   ELSE
       // ruch czarnych
       // 
       //ruch po skosie 
       #wykonuj_petle := TRUE;
       #poz_temp := #hetman.pozycja;
       WHILE #wykonuj_petle DO
           #poz_temp.x += 1;
           #poz_temp.y += 1;
           IF "sprawdz_czy_na_szachownicy"(#poz_temp) = true THEN
               IF "sprawdz_czy_wolne"(pozycja := #poz_temp, szachownica := #szachownica) = true THEN
                   IF "sprawdz_czy_ruch_możliwy"(figura := #hetman, szachownica := #szachownica, pozycja := #poz_temp) = true  THEN
                       #hetman.mozliwe_ruchy[#indeks_mozliwych_ruchow] := #poz_temp;
                       #indeks_mozliwych_ruchow += 1;
                   END_IF;
               ELSIF "sprawdz_czy_zajete"(pozycja := #poz_temp, szachownica := #szachownica) = 2 THEN
                   IF "sprawdz_czy_ruch_możliwy"(figura := #hetman, szachownica := #szachownica, pozycja := #poz_temp) = true  THEN
                       #hetman.mozliwe_ruchy[#indeks_mozliwych_ruchow] := #poz_temp;
                       #indeks_mozliwych_ruchow += 1;
                       #wykonuj_petle := false;
                   END_IF;
               ELSE
                   #wykonuj_petle := false;
               END_IF;
           ELSE
               #wykonuj_petle := false;
           END_IF;
       END_WHILE;
       #wykonuj_petle := TRUE;
       #poz_temp := #hetman.pozycja;
       WHILE #wykonuj_petle DO
           #poz_temp.x += 1;
           #poz_temp.y -= 1;
           IF "sprawdz_czy_na_szachownicy"(#poz_temp) = true THEN
               IF "sprawdz_czy_wolne"(pozycja := #poz_temp, szachownica := #szachownica) = true THEN
                   IF "sprawdz_czy_ruch_możliwy"(figura := #hetman, szachownica := #szachownica, pozycja := #poz_temp) = true  THEN
                       #hetman.mozliwe_ruchy[#indeks_mozliwych_ruchow] := #poz_temp;
                       #indeks_mozliwych_ruchow += 1;
                   END_IF;
               ELSIF "sprawdz_czy_zajete"(pozycja := #poz_temp, szachownica := #szachownica) = 2 THEN
                   IF "sprawdz_czy_ruch_możliwy"(figura := #hetman, szachownica := #szachownica, pozycja := #poz_temp) = true  THEN
                       #hetman.mozliwe_ruchy[#indeks_mozliwych_ruchow] := #poz_temp;
                       #indeks_mozliwych_ruchow += 1;
                       #wykonuj_petle := false;
                   END_IF;
               ELSE
                   #wykonuj_petle := false;
               END_IF;
           ELSE
               #wykonuj_petle := false;
           END_IF;
       END_WHILE;
       #wykonuj_petle := TRUE;
       #poz_temp := #hetman.pozycja;
       WHILE #wykonuj_petle DO
           #poz_temp.x -= 1;
           #poz_temp.y += 1;
           IF "sprawdz_czy_na_szachownicy"(#poz_temp) = true THEN
               IF "sprawdz_czy_wolne"(pozycja := #poz_temp, szachownica := #szachownica) = true THEN
                   IF "sprawdz_czy_ruch_możliwy"(figura := #hetman, szachownica := #szachownica, pozycja := #poz_temp) = true  THEN
                       #hetman.mozliwe_ruchy[#indeks_mozliwych_ruchow] := #poz_temp;
                       #indeks_mozliwych_ruchow += 1;
                   END_IF;
               ELSIF "sprawdz_czy_zajete"(pozycja := #poz_temp, szachownica := #szachownica) = 2 THEN
                   IF "sprawdz_czy_ruch_możliwy"(figura := #hetman, szachownica := #szachownica, pozycja := #poz_temp) = true  THEN
                       #hetman.mozliwe_ruchy[#indeks_mozliwych_ruchow] := #poz_temp;
                       #indeks_mozliwych_ruchow += 1;
                       #wykonuj_petle := false;
                   END_IF;
               ELSE
                   #wykonuj_petle := false;
               END_IF;
           ELSE
               #wykonuj_petle := false;
           END_IF;
       END_WHILE;
       #wykonuj_petle := TRUE;
       #poz_temp := #hetman.pozycja;
       WHILE #wykonuj_petle DO
           #poz_temp.x -= 1;
           #poz_temp.y -= 1;
           IF "sprawdz_czy_na_szachownicy"(#poz_temp) = true THEN
               IF "sprawdz_czy_wolne"(pozycja := #poz_temp, szachownica := #szachownica) = true THEN
                   IF "sprawdz_czy_ruch_możliwy"(figura := #hetman, szachownica := #szachownica, pozycja := #poz_temp) = true  THEN
                       #hetman.mozliwe_ruchy[#indeks_mozliwych_ruchow] := #poz_temp;
                       #indeks_mozliwych_ruchow += 1;
                   END_IF;
               ELSIF "sprawdz_czy_zajete"(pozycja := #poz_temp, szachownica := #szachownica) = 2 THEN
                   IF "sprawdz_czy_ruch_możliwy"(figura := #hetman, szachownica := #szachownica, pozycja := #poz_temp) = true  THEN
                       #hetman.mozliwe_ruchy[#indeks_mozliwych_ruchow] := #poz_temp;
                       #indeks_mozliwych_ruchow += 1;
                       #wykonuj_petle := false;
                   END_IF;
               ELSE
                   #wykonuj_petle := false;
               END_IF;
           ELSE
               #wykonuj_petle := false;
           END_IF;
       END_WHILE;
       //ruch poziomo i pionowo
       #wykonuj_petle := TRUE;
       #poz_temp := #hetman.pozycja;
       WHILE #wykonuj_petle DO
           #poz_temp.x += 1;
           #poz_temp.y += 0;
           IF "sprawdz_czy_na_szachownicy"(#poz_temp) = true THEN
               IF "sprawdz_czy_wolne"(pozycja := #poz_temp, szachownica := #szachownica) = true THEN
                   IF "sprawdz_czy_ruch_możliwy"(figura := #hetman, szachownica := #szachownica, pozycja := #poz_temp) = true   THEN
                       #hetman.mozliwe_ruchy[#indeks_mozliwych_ruchow] := #poz_temp;
                       #indeks_mozliwych_ruchow += 1;
                   END_IF;
               ELSIF "sprawdz_czy_zajete"(pozycja := #poz_temp, szachownica := #szachownica) = 2 THEN
                   IF "sprawdz_czy_ruch_możliwy"(figura := #hetman, szachownica := #szachownica, pozycja := #poz_temp) = true   THEN
                       #hetman.mozliwe_ruchy[#indeks_mozliwych_ruchow] := #poz_temp;
                       #indeks_mozliwych_ruchow += 1;
                       #wykonuj_petle := false;
                   END_IF;
               ELSE
                   #wykonuj_petle := false;
               END_IF;
           ELSE
               #wykonuj_petle := false;
           END_IF;
       END_WHILE;
       #wykonuj_petle := TRUE;
       #poz_temp := #hetman.pozycja;
       WHILE #wykonuj_petle DO
           #poz_temp.x += 0;
           #poz_temp.y += 1;
           IF "sprawdz_czy_na_szachownicy"(#poz_temp) = true THEN
               IF "sprawdz_czy_wolne"(pozycja := #poz_temp, szachownica := #szachownica) = true THEN
                   IF "sprawdz_czy_ruch_możliwy"(figura := #hetman, szachownica := #szachownica, pozycja := #poz_temp) = true   THEN
                       #hetman.mozliwe_ruchy[#indeks_mozliwych_ruchow] := #poz_temp;
                       #indeks_mozliwych_ruchow += 1;
                   END_IF;
               ELSIF "sprawdz_czy_zajete"(pozycja := #poz_temp, szachownica := #szachownica) = 2 THEN
                   IF "sprawdz_czy_ruch_możliwy"(figura := #hetman, szachownica := #szachownica, pozycja := #poz_temp) = true   THEN
                       #hetman.mozliwe_ruchy[#indeks_mozliwych_ruchow] := #poz_temp;
                       #indeks_mozliwych_ruchow += 1;
                       #wykonuj_petle := false;
                   END_IF;
               ELSE
                   #wykonuj_petle := false;
               END_IF;
           ELSE
               #wykonuj_petle := false;
           END_IF;
       END_WHILE;
       #wykonuj_petle := TRUE;
       #poz_temp := #hetman.pozycja;
       WHILE #wykonuj_petle DO
           #poz_temp.x += -1;
           #poz_temp.y += 0;
           IF "sprawdz_czy_na_szachownicy"(#poz_temp) = true THEN
               IF "sprawdz_czy_wolne"(pozycja := #poz_temp, szachownica := #szachownica) = true THEN
                   IF "sprawdz_czy_ruch_możliwy"(figura := #hetman, szachownica := #szachownica, pozycja := #poz_temp) = true  THEN
                       #hetman.mozliwe_ruchy[#indeks_mozliwych_ruchow] := #poz_temp;
                       #indeks_mozliwych_ruchow += 1;
                   END_IF;
               ELSIF "sprawdz_czy_zajete"(pozycja := #poz_temp, szachownica := #szachownica) = 2 THEN
                   IF "sprawdz_czy_ruch_możliwy"(figura := #hetman, szachownica := #szachownica, pozycja := #poz_temp) = true  THEN
                       #hetman.mozliwe_ruchy[#indeks_mozliwych_ruchow] := #poz_temp;
                       #indeks_mozliwych_ruchow += 1;
                       #wykonuj_petle := false;
                   END_IF;
               ELSE
                   #wykonuj_petle := false;
               END_IF;
           ELSE
               #wykonuj_petle := false;
           END_IF;
       END_WHILE;
       #wykonuj_petle := TRUE;
       #poz_temp := #hetman.pozycja;
       WHILE #wykonuj_petle DO
           #poz_temp.x += 0;
           #poz_temp.y += -1;
           IF "sprawdz_czy_na_szachownicy"(#poz_temp) = true THEN
               IF "sprawdz_czy_wolne"(pozycja := #poz_temp, szachownica := #szachownica) = true THEN
                   IF "sprawdz_czy_ruch_możliwy"(figura := #hetman, szachownica := #szachownica, pozycja := #poz_temp) = true  THEN
                       #hetman.mozliwe_ruchy[#indeks_mozliwych_ruchow] := #poz_temp;
                       #indeks_mozliwych_ruchow += 1;
                   END_IF;
               ELSIF "sprawdz_czy_zajete"(pozycja := #poz_temp, szachownica := #szachownica) = 2 THEN
                   IF ("sprawdz_czy_ruch_możliwy"(figura := #hetman, szachownica := #szachownica, pozycja := #poz_temp) = true )  THEN
                       #hetman.mozliwe_ruchy[#indeks_mozliwych_ruchow] := #poz_temp;
                       #indeks_mozliwych_ruchow += 1;
                       #wykonuj_petle := false;
                   END_IF;
               ELSE
                   #wykonuj_petle := false;
               END_IF;
           ELSE
               #wykonuj_petle := false;
           END_IF;
       END_WHILE;
   END_IF;
   #sprawdz_ruch_hetmana := #indeks_mozliwych_ruchow;
END_FUNCTION

FUNCTION "sprawdz_czy_na_szachownicy" : Bool   // FC15, SCL
{ S7_Optimized_Access := 'TRUE' }
VERSION : 0.1
   VAR_INPUT
      pozycja : "Pozycja";   // pozycja do sprawdzenia
   END_VAR
BEGIN
   IF (#pozycja.x > 8 OR #pozycja.x < 1 OR #pozycja.y > 8 OR #pozycja.y < 1) THEN
       #sprawdz_czy_na_szachownicy := 0;
   ELSE
       #sprawdz_czy_na_szachownicy := 1;
   END_IF;
END_FUNCTION

FUNCTION "sprawdz_czy_ruch_możliwy" : Bool   // FC16, SCL
{ S7_Optimized_Access := 'TRUE' }
VERSION : 0.1
   VAR_INPUT
      szachownica : "Szachownica";
      pozycja : "Pozycja";
   END_VAR
   VAR_IN_OUT
      figura : "Figura";
   END_VAR
   VAR_TEMP
      szachownica_temp : "Szachownica";
      i : Int;
   END_VAR
BEGIN
   #szachownica_temp := #szachownica;

   "wykonanie_ruchu"(szachownica:=#szachownica_temp,
                     figura:=#figura,
                     pozycja:=#pozycja);


   #sprawdz_czy_ruch_możliwy:=  NOT "sprawdz_czy_szach"(tura_bool:="Status_rozgrywki".tura_bool,
                       szachownica:=#szachownica_temp);
END_FUNCTION

(* ===== HMI "HMI_RT_1" =====
system functions are stored by id; their names below are inferred from use
connection "HMI_Connection_1": ETHERNET, S7_1500_OMS

HMI tags "Status figur"
   "status" : Array [0..63] of Int = PLC StatusyHMI."statusy figur" AT %DB1.DBX8.0, 100 ms
   "press1" : DWord AT %DB1.DBD4, 100 ms
   "press2" : DWord AT %DB1.DBD0, 100 ms
   "buttons_visibility" : Array [0..63] of Bool = PLC StatusyHMI."przyciski widocznosc" AT %DB1.DBX136.0, 100 ms

HMI tags "Status gry"
   "szach_biale" : Bool = PLC Status_rozgrywki.szach_biale, 100 ms
   "szach_czarne" : Bool = PLC Status_rozgrywki.szach_czarne, 100 ms
   "szachmat_biale" : Bool = PLC Status_rozgrywki.szachmat_biale, 100 ms
   "szachmat_czarne" : Bool = PLC Status_rozgrywki.szachmat_czarne, 100 ms
   "tura_bool" : Bool = PLC Status_rozgrywki.tura_bool, 100 ms
   "inicjalizacja" : Bool = PLC Status_rozgrywki.inicjalizacja AT %DB1.DBX0.0, 100 ms
   "status_zakonczenia_gry" : Bool = PLC Status_rozgrywki.status_zakonczenia_gry AT %DB1.DBX0.0, 100 ms
   "komunikat_koniec_gry" : Int = PLC Status_rozgrywki.komunikat_koniec_gry AT %DB1.DBX0.0, 100 ms
   "remis" : Bool = PLC Status_rozgrywki.remis AT %DB1.DBX0.0, 100 ms

text list "tura": 1 'Tura białe'; 0 'Tura czarne'

text list "komunikat_koniec": 0 'Wygrały białe !'; 1 'Wygrały czarne !'; 2 'Remis'

graphic list "Chess": 0 'wpawn'; 1 'wbishop'; 2 'whorse'; 3 'wtower'; 4 'wqueen'; 5 'wking'; 6 'bpawn'; 7 'bbishop'; 8 'bhorse'; 9 'btower'; 10 'bqueen'; 11 'bking'; 12 'blank'

screen "Root screen" 800x480, template "Template_1"
   TextField "HmiScreenItemData_1" at 72,225 size 576x25; Text 'Welcome to HMI_1 (TP700 Comfort)!'
   Button "HmiScreenItemData" at 36,36 size 159x47; TextOn 'Game Screen'; TextOff 'Game Screen'; PictureOn "Navigates to Game Screen for TP700 Comfort 14.0.1.0"; PictureOff "Navigates to Game Screen for TP700 Comfort 14.0.1.0"
      on Release: ActivateScreen("GameScreen", 0)

screen "GameScreen" 800x480, template "Template_1"
   Button "Back" at 1,8 size 159x47; TextOn 'Back'; TextOff 'Back'
      on Release: ActivateScreen("Root screen", 0)
   Button "Back_3" at 2,149 size 159x47; TextOn 'Back'; TextOff 'Back'; TextList "tura"
      ProcessValue <- "tura_bool"
   Button "Back_1" at 2,60 size 159x47; TextOn 'Back'; TextOff 'Restart'
      on Click: SetBit("inicjalizacja")
   TextField "Text field_1" at 616,60 size 70x28; Text 'Szach'
      Visibility <- "szach_czarne"
   TextField "Text field_2" at 616,409 size 70x28; Text 'Szach'
      Visibility <- "szach_biale"
   Group "Group" at 194,49 size 400x400
   Group "figury" at 194,49 size 400x400; PictureList "Chess"
   Button "Button_1" at 194,49 size 50x50; TextOff 'Text'
      on Press: function_c82f6f27("press1", 0)
      Visibility <- "[0]"
      Appearance <- "press1"
   Button "Button_2" at 244,49 size 50x50; TextOff 'Text'
      on Press: function_c82f6f27("press1", 1)
      Appearance <- "press1"
      Visibility <- "[1]"
   Button "Button_3" at 294,49 size 50x50; TextOff 'Text'
      on Press: function_c82f6f27("press1", 2)
      Appearance <- "press1"
      Visibility <- "[2]"
   Button "Button_4" at 344,49 size 50x50; TextOff 'Text'
      on Press: function_c82f6f27("press1", 3)
      Appearance <- "press1"
      Visibility <- "[3]"
   Button "Button_5" at 394,49 size 50x50; TextOff 'Text'
      on Press: function_c82f6f27("press1", 4)
      Appearance <- "press1"
      Visibility <- "[4]"
   Button "Button_6" at 444,49 size 50x50; TextOff 'Text'
      on Press: function_c82f6f27("press1", 5)
      Appearance <- "press1"
      Visibility <- "[5]"
   Button "Button_7" at 494,49 size 49x50; TextOff 'Text'
      on Press: function_c82f6f27("press1", 6)
      Appearance <- "press1"
      Visibility <- "[6]"
   Button "Button_8" at 544,49 size 50x50; TextOff 'Text'
      on Press: function_c82f6f27("press1", 7)
      Appearance <- "press1"
      Visibility <- "[7]"
   Button "Button_9" at 194,99 size 50x50; TextOff 'Text'
      on Press: function_c82f6f27("press1", 8)
      Appearance <- "press1"
      Visibility <- "[8]"
   Button "Button_10" at 244,99 size 50x50; TextOff 'Text'
      on Press: function_c82f6f27("press1", 9)
      Appearance <- "press1"
      Visibility <- "[9]"
   Button "Button_11" at 294,99 size 50x50; TextOff 'Text'
      on Press: function_c82f6f27("press1", 10)
      Appearance <- "press1"
      Visibility <- "[10]"
   Button "Button_12" at 344,99 size 50x50; TextOff 'Text'
      on Press: function_c82f6f27("press1", 11)
      Appearance <- "press1"
      Visibility <- "[11]"
   Button "Button_13" at 394,99 size 50x50; TextOff 'Text'
      on Press: function_c82f6f27("press1", 12)
      Appearance <- "press1"
      Visibility <- "[12]"
   Button "Button_14" at 444,99 size 50x50; TextOff 'Text'
      on Press: function_c82f6f27("press1", 13)
      Appearance <- "press1"
      Visibility <- "[13]"
   Button "Button_15" at 494,99 size 50x50; TextOff 'Text'
      on Press: function_c82f6f27("press1", 14)
      Appearance <- "press1"
      Visibility <- "[14]"
   Button "Button_16" at 544,99 size 50x50; TextOff 'Text'
      on Press: function_c82f6f27("press1", 15)
      Appearance <- "press1"
      Visibility <- "[15]"
   Button "Button_17" at 194,149 size 50x50; TextOff 'Text'
      on Press: function_c82f6f27("press1", 16)
      Appearance <- "press1"
      Visibility <- "[16]"
   Button "Button_18" at 244,149 size 50x50; TextOff 'Text'
      on Press: function_c82f6f27("press1", 17)
      Appearance <- "press1"
      Visibility <- "[17]"
   Button "Button_19" at 294,149 size 50x50; TextOff 'Text'
      on Press: function_c82f6f27("press1", 18)
      Appearance <- "press1"
      Visibility <- "[18]"
   Button "Button_20" at 344,149 size 50x50; TextOff 'Text'
      on Press: function_c82f6f27("press1", 19)
      Appearance <- "press1"
      Visibility <- "[19]"
   Button "Button_21" at 394,149 size 50x50; TextOff 'Text'
      on Press: function_c82f6f27("press1", 20)
      Appearance <- "press1"
      Visibility <- "[20]"
   Button "Button_22" at 444,149 size 50x50; TextOff 'Text'
      on Press: function_c82f6f27("press1", 21)
      Appearance <- "press1"
      Visibility <- "[21]"
   Button "Button_23" at 494,149 size 50x50; TextOff 'Text'
      on Press: function_c82f6f27("press1", 22)
      Appearance <- "press1"
      Visibility <- "[22]"
   Button "Button_24" at 544,149 size 50x50; TextOff 'Text'
      on Press: function_c82f6f27("press1", 23)
      Appearance <- "press1"
      Visibility <- "[23]"
   Button "Button_25" at 194,199 size 50x50; TextOff 'Text'
      on Press: function_c82f6f27("press1", 24)
      Appearance <- "press1"
      Visibility <- "[24]"
   Button "Button_26" at 244,199 size 50x50; TextOff 'Text'
      on Press: function_c82f6f27("press1", 25)
      Appearance <- "press1"
      Visibility <- "[25]"
   Button "Button_27" at 294,199 size 50x50; TextOff 'Text'
      on Press: function_c82f6f27("press1", 26)
      Appearance <- "press1"
      Visibility <- "[26]"
   Button "Button_28" at 344,199 size 50x50; TextOff 'Text'
      on Press: function_c82f6f27("press1", 27)
      Appearance <- "press1"
      Visibility <- "[27]"
   Button "Button_29" at 394,199 size 50x50; TextOff 'Text'
      on Press: function_c82f6f27("press1", 28)
      Appearance <- "press1"
      Visibility <- "[28]"
   Button "Button_30" at 444,199 size 50x50; TextOff 'Text'
      on Press: function_c82f6f27("press1", 29)
      Appearance <- "press1"
      Visibility <- "[29]"
   Button "Button_31" at 494,199 size 50x50; TextOff 'Text'
      on Press: function_c82f6f27("press1", 30)
      Appearance <- "press1"
      Visibility <- "[30]"
   Button "Button_32" at 544,199 size 50x50; TextOff 'Text'
      on Press: function_c82f6f27("press1", 31)
      Appearance <- "press1"
      Visibility <- "[31]"
   Button "Button_33" at 194,249 size 50x50; TextOff 'Text'
      on Press: function_c82f6f27("press2", 0)
      Visibility <- "[32]"
   Button "Button_34" at 244,249 size 50x50; TextOff 'Text'
      on Press: function_c82f6f27("press2", 1)
      Visibility <- "[33]"
   Button "Button_35" at 294,249 size 50x50; TextOff 'Text'
      on Press: function_c82f6f27("press2", 2)
      Visibility <- "[34]"
   Button "Button_36" at 344,249 size 50x50; TextOff 'Text'
      on Press: function_c82f6f27("press2", 3)
      Visibility <- "[35]"
   Button "Button_37" at 394,249 size 50x50; TextOff 'Text'
      on Press: function_c82f6f27("press2", 4)
      Visibility <- "[36]"
   Button "Button_38" at 444,249 size 50x50; TextOff 'Text'
      on Press: function_c82f6f27("press2", 5)
      Visibility <- "[37]"
   Button "Button_39" at 494,249 size 50x50; TextOff 'Text'
      on Press: function_c82f6f27("press2", 6)
      Visibility <- "[38]"
   Button "Button_40" at 544,249 size 50x50; TextOff 'Text'
      on Press: function_c82f6f27("press2", 7)
      Visibility <- "[39]"
   Button "Button_41" at 194,299 size 50x50; TextOff 'Text'
      on Press: function_c82f6f27("press2", 8)
      Visibility <- "[40]"
   Button "Button_42" at 244,299 size 50x50; TextOff 'Text'
      on Press: function_c82f6f27("press2", 9)
      Visibility <- "[41]"
   Button "Button_43" at 294,299 size 50x50; TextOff 'Text'
      on Press: function_c82f6f27("press2", 10)
      Visibility <- "[42]"
   Button "Button_44" at 344,299 size 50x50; TextOff 'Text'
      on Press: function_c82f6f27("press2", 11)
      Visibility <- "[43]"
   Button "Button_45" at 394,299 size 50x50; TextOff 'Text'
      on Press: function_c82f6f27("press2", 12)
      Visibility <- "[44]"
   Button "Button_46" at 444,299 size 50x50; TextOff 'Text'
      on Press: function_c82f6f27("press2", 13)
      Visibility <- "[45]"
   Button "Button_47" at 494,299 size 50x50; TextOff 'Text'
      on Press: function_c82f6f27("press2", 14)
      Visibility <- "[46]"
   Button "Button_48" at 545,303 size 50x50; TextOff 'Text'
      on Press: function_c82f6f27("press2", 15)
      Visibility <- "[47]"
   Button "Button_49" at 194,349 size 50x50; TextOff 'Text'
      on Press: function_c82f6f27("press2", 16)
      Visibility <- "[48]"
   Button "Button_50" at 244,349 size 50x50; TextOff 'Text'
      on Press: function_c82f6f27("press2", 17)
      Visibility <- "[49]"
   Button "Button_51" at 294,349 size 50x50; TextOff 'Text'
      on Press: function_c82f6f27("press2", 18)
      Visibility <- "[50]"
   Button "Button_52" at 344,349 size 50x50; TextOff 'Text'
      on Press: function_c82f6f27("press2", 19)
      Visibility <- "[51]"
   Button "Button_53" at 394,349 size 50x50; TextOff 'Text'
      on Press: function_c82f6f27("press2", 20)
      Visibility <- "[52]"
   Button "Button_54" at 444,349 size 50x50; TextOff 'Text'
      on Press: function_c82f6f27("press2", 21)
      Visibility <- "[53]"
   Button "Button_55" at 494,349 size 50x50; TextOff 'Text'
      on Press: function_c82f6f27("press2", 22)
      Visibility <- "[54]"
   Button "Button_56" at 544,349 size 50x50; TextOff 'Text'
      on Press: function_c82f6f27("press2", 23)
      Visibility <- "[55]"
   Button "Button_57" at 194,399 size 50x50; TextOff 'Text'
      on Press: function_c82f6f27("press2", 24)
      Visibility <- "[56]"
   Button "Button_58" at 244,399 size 50x50; TextOff 'Text'
      on Press: function_c82f6f27("press2", 25)
      Visibility <- "[57]"
   Button "Button_59" at 294,399 size 50x50; TextOff 'Text'
      on Press: function_c82f6f27("press2", 26)
      Visibility <- "[58]"
   Button "Button_60" at 344,399 size 50x50; TextOff 'Text'
      on Press: function_c82f6f27("press2", 27)
      Visibility <- "[59]"
   Button "Button_61" at 394,399 size 50x50; TextOff 'Text'
      on Press: function_c82f6f27("press2", 28)
      Visibility <- "[60]"
   Button "Button_62" at 444,399 size 50x50; TextOff 'Text'
      on Press: function_c82f6f27("press2", 29)
      Visibility <- "[61]"
   Button "Button_63" at 494,399 size 50x50; TextOff 'Text'
      on Press: function_c82f6f27("press2", 30)
      Visibility <- "[62]"
   Button "Button_64" at 544,399 size 50x50; TextOff 'Text'
      on Press: function_c82f6f27("press2", 31)
      Visibility <- "[63]"
   Rectangle "Rectangle_2" at 194,99 size 50x50
      Appearance <- "press1"
   Rectangle "Rectangle_3" at 194,199 size 50x50
      Appearance <- "press1"
   Rectangle "Rectangle_4" at 194,299 size 50x50
      Appearance <- "press2"
   Rectangle "Rectangle_5" at 194,399 size 50x50
      Appearance <- "press2"
   Rectangle "Rectangle_6" at 244,49 size 50x50
      Appearance <- "press1"
   Rectangle "Rectangle_7" at 244,149 size 50x50
      Appearance <- "press1"
   Rectangle "Rectangle_8" at 244,249 size 50x50
      Appearance <- "press2"
   Rectangle "Rectangle_9" at 244,349 size 50x50
      Appearance <- "press2"
   Rectangle "Rectangle_10" at 294,99 size 50x50
      Appearance <- "press1"
   Rectangle "Rectangle_11" at 294,199 size 50x50
      Appearance <- "press1"
   Rectangle "Rectangle_12" at 294,299 size 50x50
      Appearance <- "press2"
   Rectangle "Rectangle_13" at 293,399 size 50x50
      Appearance <- "press2"
   Rectangle "Rectangle_14" at 344,49 size 50x50
      Appearance <- "press1"
   Rectangle "Rectangle_15" at 344,149 size 50x50
      Appearance <- "press1"
   Rectangle "Rectangle_16" at 344,249 size 50x50
      Appearance <- "press2"
   Rectangle "Rectangle_17" at 344,349 size 50x50
      Appearance <- "press2"
   Rectangle "Rectangle_18" at 394,99 size 50x50
      Appearance <- "press1"
   Rectangle "Rectangle_19" at 394,199 size 50x50
      Appearance <- "press1"
   Rectangle "Rectangle_20" at 394,299 size 50x50
      Appearance <- "press2"
   Rectangle "Rectangle_21" at 394,399 size 50x50
      Appearance <- "press2"
   Rectangle "Rectangle_22" at 444,49 size 50x50
      Appearance <- "press1"
   Rectangle "Rectangle_23" at 444,149 size 50x50
      Appearance <- "press1"
   Rectangle "Rectangle_24" at 444,249 size 50x50
      Appearance <- "press2"
   Rectangle "Rectangle_25" at 444,349 size 50x50
      Appearance <- "press2"
   Rectangle "Rectangle_26" at 494,99 size 50x50
      Appearance <- "press1"
   Rectangle "Rectangle_27" at 494,199 size 50x50
      Appearance <- "press1"
   Rectangle "Rectangle_28" at 494,299 size 50x50
      Appearance <- "press2"
   Rectangle "Rectangle_29" at 494,399 size 50x50
      Appearance <- "press2"
   Rectangle "Rectangle_30" at 544,49 size 50x50
      Appearance <- "press1"
   Rectangle "Rectangle_31" at 544,149 size 50x50
      Appearance <- "press1"
   Rectangle "Rectangle_32" at 544,249 size 50x50
      Appearance <- "press2"
   Rectangle "Rectangle_33" at 544,349 size 50x50
      Appearance <- "press2"
   Rectangle "Rectangle_1" at 194,49 size 50x50
      Appearance <- "press1"
   Rectangle "Rectangle_34" at 294,49 size 50x50
      Appearance <- "press1"
   Rectangle "Rectangle_35" at 394,49 size 50x50
      Appearance <- "press1"
   Rectangle "Rectangle_36" at 494,49 size 50x50
      Appearance <- "press1"
   Rectangle "Rectangle_37" at 244,99 size 50x50
      Appearance <- "press1"
   Rectangle "Rectangle_38" at 344,99 size 50x50
      Appearance <- "press1"
   Rectangle "Rectangle_39" at 444,99 size 50x50
      Appearance <- "press1"
   Rectangle "Rectangle_40" at 544,99 size 50x50
      Appearance <- "press1"
   Rectangle "Rectangle_41" at 194,149 size 50x50
      Appearance <- "press1"
   Rectangle "Rectangle_42" at 294,149 size 50x50
      Appearance <- "press1"
   Rectangle "Rectangle_43" at 394,149 size 50x50
      Appearance <- "press1"
   Rectangle "Rectangle_44" at 494,149 size 50x50
      Appearance <- "press1"
   Rectangle "Rectangle_45" at 244,199 size 50x50
      Appearance <- "press1"
   Rectangle "Rectangle_46" at 344,199 size 50x50
      Appearance <- "press1"
   Rectangle "Rectangle_47" at 444,199 size 50x50
      Appearance <- "press1"
   Rectangle "Rectangle_48" at 544,199 size 50x50
      Appearance <- "press1"
   Rectangle "Rectangle_49" at 194,249 size 50x50
      Appearance <- "press2"
   Rectangle "Rectangle_50" at 294,249 size 50x50
      Appearance <- "press2"
   Rectangle "Rectangle_51" at 394,249 size 50x50
      Appearance <- "press2"
   Rectangle "Rectangle_52" at 494,249 size 50x50
      Appearance <- "press2"
   Rectangle "Rectangle_53" at 244,299 size 50x50
      Appearance <- "press2"
   Rectangle "Rectangle_54" at 344,299 size 50x50
      Appearance <- "press2"
   Rectangle "Rectangle_55" at 444,299 size 50x50
      Appearance <- "press2"
   Rectangle "Rectangle_56" at 544,299 size 50x50
      Appearance <- "press2"
   Rectangle "Rectangle_57" at 194,349 size 50x50
      Appearance <- "press2"
   Rectangle "Rectangle_58" at 294,349 size 50x50
      Appearance <- "press2"
   Rectangle "Rectangle_59" at 394,349 size 50x50
      Appearance <- "press2"
   Rectangle "Rectangle_60" at 494,349 size 50x50
      Appearance <- "press2"
   Rectangle "Rectangle_61" at 244,399 size 50x50
      Appearance <- "press2"
   Rectangle "Rectangle_62" at 344,399 size 50x50
      Appearance <- "press2"
   Rectangle "Rectangle_63" at 444,399 size 50x50
      Appearance <- "press2"
   Rectangle "Rectangle_64" at 544,399 size 50x50
      Appearance <- "press2"
   GraphicIOField "1" at 194,49 size 50x50; PictureList "Chess"
      ProcessValue <- "[0]"
   GraphicIOField "2" at 244,49 size 50x50; PictureList "Chess"
      ProcessValue <- "[1]"
   GraphicIOField "3" at 296,49 size 50x50; PictureList "Chess"
      ProcessValue <- "[2]"
   GraphicIOField "4" at 344,49 size 50x50; PictureList "Chess"
      ProcessValue <- "[3]"
   GraphicIOField "5" at 394,49 size 50x50; PictureList "Chess"
      ProcessValue <- "[4]"
   GraphicIOField "6" at 444,49 size 50x50; PictureList "Chess"
      ProcessValue <- "[5]"
   GraphicIOField "7" at 494,49 size 50x50; PictureList "Chess"
      ProcessValue <- "[6]"
   GraphicIOField "8" at 544,49 size 50x50; PictureList "Chess"
      ProcessValue <- "[7]"
   GraphicIOField "9" at 194,99 size 50x50; PictureList "Chess"
      ProcessValue <- "[8]"
   GraphicIOField "10" at 244,99 size 50x50; PictureList "Chess"
      ProcessValue <- "[9]"
   GraphicIOField "11" at 296,99 size 50x50; PictureList "Chess"
      ProcessValue <- "[10]"
   GraphicIOField "12" at 344,99 size 50x50; PictureList "Chess"
      ProcessValue <- "[11]"
   GraphicIOField "13" at 394,99 size 50x50; PictureList "Chess"
      ProcessValue <- "[12]"
   GraphicIOField "14" at 444,99 size 50x50; PictureList "Chess"
      ProcessValue <- "[13]"
   GraphicIOField "15" at 494,99 size 50x50; PictureList "Chess"
      ProcessValue <- "[14]"
   GraphicIOField "16" at 544,99 size 50x50; PictureList "Chess"
      ProcessValue <- "[15]"
   GraphicIOField "17" at 194,149 size 50x50; PictureList "Chess"
      ProcessValue <- "[16]"
   GraphicIOField "18" at 244,149 size 50x50; PictureList "Chess"
      ProcessValue <- "[17]"
   GraphicIOField "19" at 296,149 size 50x50; PictureList "Chess"
      ProcessValue <- "[18]"
   GraphicIOField "20" at 344,149 size 50x50; PictureList "Chess"
      ProcessValue <- "[19]"
   GraphicIOField "21" at 394,149 size 50x50; PictureList "Chess"
      ProcessValue <- "[20]"
   GraphicIOField "22" at 444,149 size 50x50; PictureList "Chess"
      ProcessValue <- "[21]"
   GraphicIOField "23" at 494,149 size 50x50; PictureList "Chess"
      ProcessValue <- "[22]"
   GraphicIOField "24" at 544,149 size 50x50; PictureList "Chess"
      ProcessValue <- "[23]"
   GraphicIOField "25" at 194,199 size 50x50; PictureList "Chess"
      ProcessValue <- "[24]"
   GraphicIOField "26" at 244,199 size 50x50; PictureList "Chess"
      ProcessValue <- "[25]"
   GraphicIOField "27" at 296,199 size 50x50; PictureList "Chess"
      ProcessValue <- "[26]"
   GraphicIOField "28" at 344,199 size 50x50; PictureList "Chess"
      ProcessValue <- "[27]"
   GraphicIOField "29" at 394,199 size 50x50; PictureList "Chess"
      ProcessValue <- "[28]"
   GraphicIOField "30" at 444,199 size 50x50; PictureList "Chess"
      ProcessValue <- "[29]"
   GraphicIOField "31" at 494,199 size 50x50; PictureList "Chess"
      ProcessValue <- "[30]"
   GraphicIOField "32" at 544,199 size 50x50; PictureList "Chess"
      ProcessValue <- "[31]"
   GraphicIOField "33" at 194,249 size 50x50; PictureList "Chess"
      ProcessValue <- "[32]"
   GraphicIOField "34" at 244,249 size 50x50; PictureList "Chess"
      ProcessValue <- "[33]"
   GraphicIOField "35" at 294,249 size 50x50; PictureList "Chess"
      ProcessValue <- "[34]"
   GraphicIOField "36" at 344,249 size 50x50; PictureList "Chess"
      ProcessValue <- "[35]"
   GraphicIOField "37" at 394,249 size 50x50; PictureList "Chess"
      ProcessValue <- "[36]"
   GraphicIOField "38" at 444,249 size 50x50; PictureList "Chess"
      ProcessValue <- "[37]"
   GraphicIOField "39" at 494,249 size 50x50; PictureList "Chess"
      ProcessValue <- "[38]"
   GraphicIOField "40" at 544,249 size 50x50; PictureList "Chess"
      ProcessValue <- "[39]"
   GraphicIOField "41" at 194,299 size 50x50; PictureList "Chess"
      ProcessValue <- "[40]"
   GraphicIOField "42" at 244,299 size 50x50; PictureList "Chess"
      ProcessValue <- "[41]"
   GraphicIOField "43" at 294,299 size 50x50; PictureList "Chess"
      ProcessValue <- "[42]"
   GraphicIOField "44" at 344,299 size 50x50; PictureList "Chess"
      ProcessValue <- "[43]"
   GraphicIOField "45" at 394,299 size 50x50; PictureList "Chess"
      ProcessValue <- "[44]"
   GraphicIOField "46" at 444,299 size 50x50; PictureList "Chess"
      ProcessValue <- "[45]"
   GraphicIOField "47" at 494,299 size 50x50; PictureList "Chess"
      ProcessValue <- "[46]"
   GraphicIOField "48" at 544,299 size 50x50; PictureList "Chess"
      ProcessValue <- "[47]"
   GraphicIOField "49" at 194,349 size 50x50; PictureList "Chess"
      ProcessValue <- "[48]"
   GraphicIOField "50" at 244,349 size 50x50; PictureList "Chess"
      ProcessValue <- "[49]"
   GraphicIOField "51" at 294,349 size 50x50; PictureList "Chess"
      ProcessValue <- "[50]"
   GraphicIOField "52" at 344,349 size 50x50; PictureList "Chess"
      ProcessValue <- "[51]"
   GraphicIOField "53" at 394,349 size 50x50; PictureList "Chess"
      ProcessValue <- "[52]"
   GraphicIOField "54" at 444,349 size 50x50; PictureList "Chess"
      ProcessValue <- "[53]"
   GraphicIOField "55" at 494,349 size 50x50; PictureList "Chess"
      ProcessValue <- "[54]"
   GraphicIOField "56" at 544,349 size 50x50; PictureList "Chess"
      ProcessValue <- "[55]"
   GraphicIOField "57" at 194,399 size 50x50; PictureList "Chess"
      ProcessValue <- "[56]"
   GraphicIOField "58" at 244,399 size 50x50; PictureList "Chess"
      ProcessValue <- "[57]"
   GraphicIOField "59" at 294,399 size 50x50; PictureList "Chess"
      ProcessValue <- "[58]"
   GraphicIOField "60" at 344,399 size 50x50; PictureList "Chess"
      ProcessValue <- "[59]"
   GraphicIOField "61" at 394,399 size 50x50; PictureList "Chess"
      ProcessValue <- "[60]"
   GraphicIOField "62" at 444,399 size 50x50; PictureList "Chess"
      ProcessValue <- "[61]"
   GraphicIOField "63" at 494,399 size 50x50; PictureList "Chess"
      ProcessValue <- "[62]"
   GraphicIOField "64" at 544,399 size 50x50; PictureList "Chess"
      ProcessValue <- "[63]"
   Rectangle "Rectangle_66" at 276,152 size 240x160
      Visibility <- "status_zakonczenia_gry"
   Button "napis" at 291,172 size 207x47; TextOn 'Back'; TextOff 'Białe wygrały !'; TextList "komunikat_koniec"
      ProcessValue <- "komunikat_koniec_gry"
      Visibility <- "status_zakonczenia_gry"
   Button "new_game" at 317,232 size 160x47; TextOn 'Back'; TextOff 'Nowa gra'
      on Click: SetBit("inicjalizacja")
      Visibility <- "status_zakonczenia_gry"
   Group "Group_1" at 276,152 size 240x160; TextList "komunikat_koniec"

Template "Template_1" 800x480
   Button "Start screen" at 720,2 size 78x58; TextOn 'Start screen'; TextOff 'Start screen'; PictureOn "NavigateHome_TP700_Comfort_TR"; PictureOff "NavigateHome_TP700_Comfort_TR"
      on Release: ActivateScreen("Root screen", 0)
   Button "Template_Button" at 720,62 size 78x58; TextOff 'Text'
   Button "Template_Button_1" at 720,122 size 78x58; TextOff 'Text'
   Button "Template_Button_2" at 720,181 size 78x58; TextOff 'Text'
   Button "Template_Button_3" at 720,241 size 78x58; TextOff 'Text'
   Button "Template_Button_4" at 720,301 size 78x58; TextOff 'Text'
   Button "Template_Button_5" at 720,360 size 78x58; TextOff 'Text'
   Button "Exit" at 720,420 size 78x58; TextOn 'Exit'; TextOff 'Exit'; PictureOn "ExitRuntime_TP700_Comfort_TR"; PictureOff "ExitRuntime_TP700_Comfort_TR"
      on Release: StopRuntime(0)

PopupScreen "białe_wygrały" 320x240
   Button "Back_3" at 80,33 size 160x47; TextOn 'Back'; TextOff 'Białe wygrały !'; TextList "Białe wygrały !"
      on Release: ActivateScreen("Root screen", 0)
      ProcessValue <- "tura_bool"
   Button "Back_1" at 85,150 size 159x47; TextOn 'Back'; TextOff 'Nowa gra'
      on Click: SetBit("inicjalizacja")

VB script "VBFunction_1"
   'Tip:
   ' 1. Use the <CTRL+SPACE> or <CTRL+I> shortcut to open a list of all objects and functions
   ' 2. Write the code using the HMI Runtime object.
   '  Example: HmiRuntime.Screens("Screen_1").
   
   
   
   ' 3. Use the <CTRL+J> shortcut to create an object reference.
   'Write the code as of this position:
       HmiRuntime.ActiveScreen.ScreenItems("Button_1").BorderColor = RGB(255, 147, 33)
*)